{attribute 'linkalways'} 
FUNCTION_BLOCK AsyncConcatStringRpcHandler IMPLEMENTS I_AsynchronousRpcHandler
VAR
END_VAR

METHOD Handle
VAR_INPUT
	Parameters : I_Deserializer;
	Response : I_AsynchronousRpcResponse;
END_VAR
VAR
	str1 : T_MAXSTRING;
	str2 : T_MAXSTRING;
	result : T_MAXSTRING;
	feedback : DeserializerFeedback;
END_VAR
IF NOT Parameters.TryGetKeyString('STR1',str1,feedback) THEN
	Response.RejectWithError('MISSING_PARAMETER',feedback.FirstError.Message);
	RETURN;
END_IF

IF NOT Parameters.TryGetKeyString('STR2',str2,feedback) THEN
	Response.RejectWithError('MISSING_PARAMETER',feedback.FirstError.Message);
	RETURN;
END_IF

result := CONCAT(str1, str2);
Response.CompleteWithString(result);
END_METHOD

END_FUNCTION_BLOCK

(* stored: Version 1.1.0.1, ProductVersion 3.1.4026.13
   POU AsyncConcatStringRpcHandler: Id {15eaf484-2338-080c-24b0-21edd7080d4a}, SpecialFunc None
   Method Handle: Id {4186d797-c671-0441-0448-472149185e0f} *)
